FUNCTION_BLOCK TestStuff
VAR_INPUT
END_VAR
VAR_OUTPUT
END_VAR
VAR
	//HydraulicCylinder : FB_HydraulicCilinderAnalog;
	mxReset: BOOL;
	mxEmStop: BOOL;
	mxAutoMode: BOOL;
	mxIsIn: BOOL;
	mxIsOut: BOOL;
	mxMovesOut: BOOL;
	mxMovesIn: BOOL;
	mxSlowMoveActive: BOOL;
	ActMeasuredPos: REAL;
	ActPos: REAL;
	mxErrorStopInPos: BOOL;
	mxErrorInit: BOOL;
	mxMoveOut: BOOL;
	mxMoveIn: BOOL;
	PositionPhysicalMeasured: REAL;
	OffsetAlarmPos: REAL;
	OffsetPos: REAL;
	EndPositionOut: REAL;
	EndPositionIn: REAL;
	Errors: ST_HydraulicErrors;
	PositionPhyisicalMeasuredOld: REAL;
	PhysicalOffsetPos: REAL;
	TestEndPos: INT;
	TestNormSpeed: INT;
	TestSlowPos: INT;
	TestSlowSpeed: INT;
	TestCreepPos: INT;
	TestCreepSpeed: REAL;
	DoThis: BOOL;
	CurrentPos: REAL;
	Blink: FB_Blink;
	//AnaTest: FB_AnalogOutMinus10_10V;
	EngInputTest: REAL;
	EngMin: REAL;
	EngMax: REAL;
	VOut: REAL;
	RawOut: INT;
END_VAR

Objects();
TestCylinder();

ACTION Objects:

END_ACTION

ACTION TestCylinder:
;
END_ACTION

END_FUNCTION_BLOCK

(* stored: Version 1.1.0.1, ProductVersion 3.1.4020.12
   POU TestStuff: Id {4aefed9b-9e84-4387-aa83-75ce843fb620}, SpecialFunc None
   Action Objects: Id {0a4bcf43-3f91-4193-be94-7e918e23ee86}
   Action TestCylinder: Id {cdf009e4-ced9-42d9-9b19-8fc81fdf51f7} *)
